Omron CX-Programmer project NewProject (CX-Programmer 9.81)

# PLC NewPLC1: CP1L M

## Program NewProgram1 (cyclic task 0)
Local symbols
Contador #0000 NUMBER
M1 3.01 BOOL
MO 3.00 BOOL
b_1 0.00 BOOL
b_reset 0.01 BOOL

### Section Section1

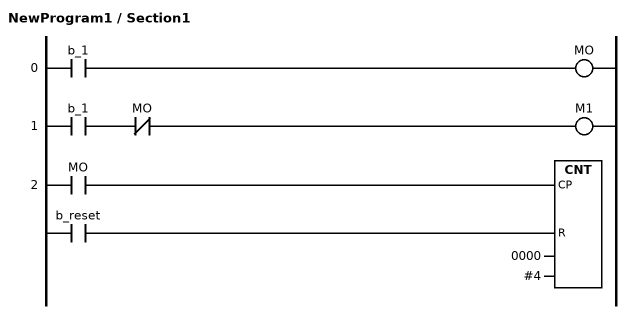
; rung 0
LD b_1
OUT MO
; rung 1
LD b_1
ANDNOT MO
OUT M1
; rung 2
LD MO
LD b_reset
CNT 0000 #4

### Section END
; rung 0
END(001)